Staubli VAL3: Queue.dtx

public num nPush
public num nPop
public num nElems
public MotionCmd buffer[15]
  [0]
    mdesc mDesc = {leave=0, reach=0}
    num nDuration
    num nSequence
    jointRx jJointRx
  [1]
    mdesc mDesc = {leave=0, reach=0}
    num nDuration
    num nSequence
    jointRx jJointRx
  [2]
    mdesc mDesc = {leave=0, reach=0}
    num nDuration
    num nSequence
    jointRx jJointRx
  [3]
    mdesc mDesc = {leave=0, reach=0}
    num nDuration
    num nSequence
    jointRx jJointRx
  [4]
    mdesc mDesc = {leave=0, reach=0}
    num nDuration
    num nSequence
    jointRx jJointRx
  [5]
    mdesc mDesc = {leave=0, reach=0}
    num nDuration
    num nSequence
    jointRx jJointRx
  [6]
    mdesc mDesc = {leave=0, reach=0}
    num nDuration
    num nSequence
    jointRx jJointRx
  [7]
    mdesc mDesc = {leave=0, reach=0}
    num nDuration
    num nSequence
    jointRx jJointRx
  [8]
    mdesc mDesc = {leave=0, reach=0}
    num nDuration
    num nSequence
    jointRx jJointRx
  [9]
    mdesc mDesc = {leave=0, reach=0}
    num nDuration
    num nSequence
    jointRx jJointRx
  [10]
    mdesc mDesc = {leave=0, reach=0}
    num nDuration
    num nSequence
    jointRx jJointRx
  [11]
    mdesc mDesc = {leave=0, reach=0}
    num nDuration
    num nSequence
    jointRx jJointRx
  [12]
    mdesc mDesc = {leave=0, reach=0}
    num nDuration
    num nSequence
    jointRx jJointRx
  [13]
    mdesc mDesc = {leave=0, reach=0}
    num nDuration
    num nSequence
    jointRx jJointRx
  [14]
    mdesc mDesc = {leave=0, reach=0}
    num nDuration
    num nSequence
    jointRx jJointRx
